PROGRAM VariableTesting
VAR
	one: MC_MoveAbsolute;
	two: MC_MoveAbsolute;
	three: MC_MoveAbsolute;
	four: MC_MoveAbsolute;
	five: MC_MoveAbsolute;
	six: MC_MoveAbsolute;
	CTU_0: CTU;
	Count: CTU;
END_VAR

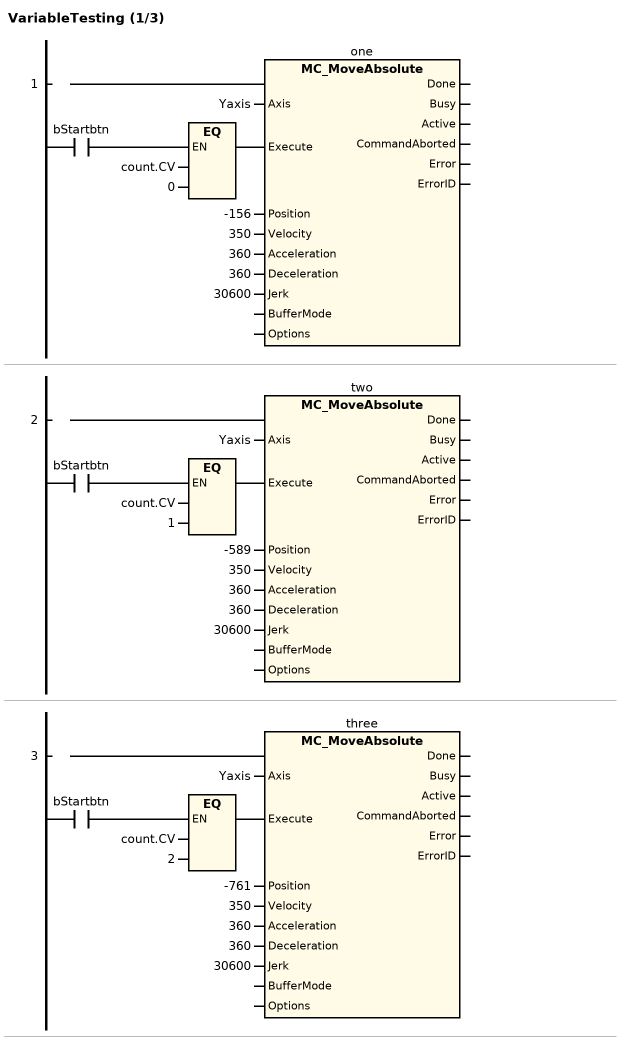
// NETWORK 1
one(
    Axis := Yaxis,
    Execute := bStartbtn AND count.CV = 0,
    Position := -156,
    Velocity := 350,
    Acceleration := 360,
    Deceleration := 360,
    Jerk := 30600); // MC_MoveAbsolute

// NETWORK 2
two(
    Axis := Yaxis,
    Execute := bStartbtn AND count.CV = 1,
    Position := -589,
    Velocity := 350,
    Acceleration := 360,
    Deceleration := 360,
    Jerk := 30600); // MC_MoveAbsolute

// NETWORK 3
three(
    Axis := Yaxis,
    Execute := bStartbtn AND count.CV = 2,
    Position := -761,
    Velocity := 350,
    Acceleration := 360,
    Deceleration := 360,
    Jerk := 30600); // MC_MoveAbsolute

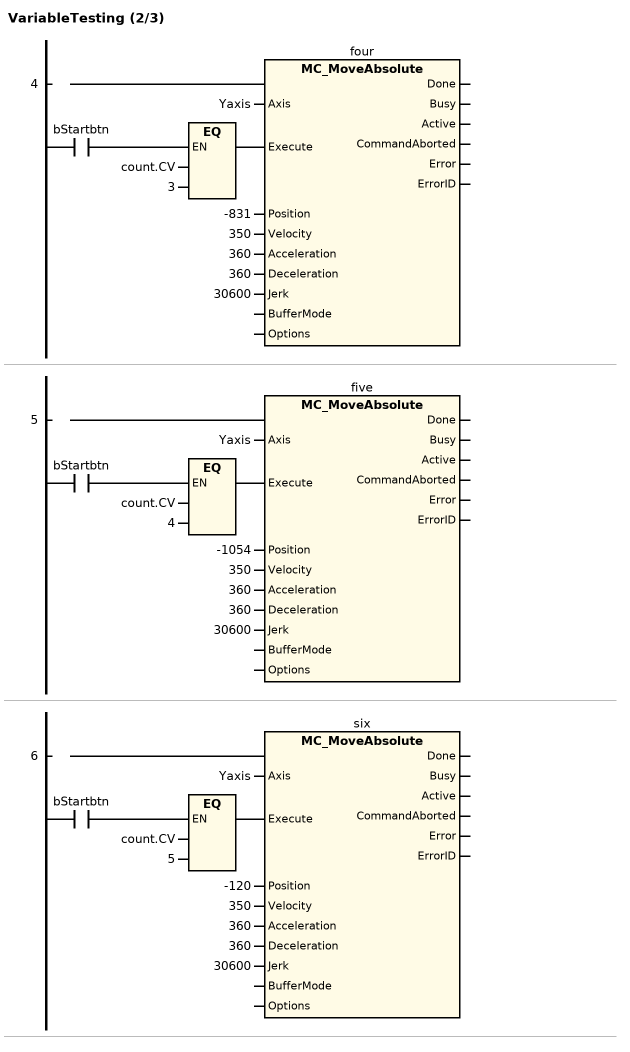
// NETWORK 4
four(
    Axis := Yaxis,
    Execute := bStartbtn AND count.CV = 3,
    Position := -831,
    Velocity := 350,
    Acceleration := 360,
    Deceleration := 360,
    Jerk := 30600); // MC_MoveAbsolute

// NETWORK 5
five(
    Axis := Yaxis,
    Execute := bStartbtn AND count.CV = 4,
    Position := -1054,
    Velocity := 350,
    Acceleration := 360,
    Deceleration := 360,
    Jerk := 30600); // MC_MoveAbsolute

// NETWORK 6
six(
    Axis := Yaxis,
    Execute := bStartbtn AND count.CV = 5,
    Position := -120,
    Velocity := 350,
    Acceleration := 360,
    Deceleration := 360,
    Jerk := 30600); // MC_MoveAbsolute

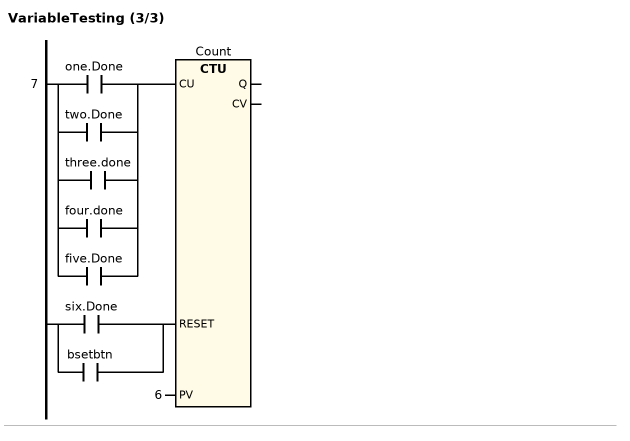
// NETWORK 7
Count(
    CU := one.Done OR two.Done OR three.done OR four.done OR five.Done,
    RESET := six.Done OR bsetbtn,
    PV := 6); // CTU

END_PROGRAM

(* stored: Version 1.1.0.1, ProductVersion 3.1.4024.12
   POU VariableTesting: Id {fb19320d-336d-452b-891f-4462dbd11eed}, SpecialFunc None *)
